(*
Searches an `I_Entity` for a `I_Receiver` component matching provided id pattern.
Result:
- Ok - Returns `I_Receiver`.
- None - Returns null.
- Err.Itf0 - Returns null, incorrect interface.
*)
FUNCTION GetReceiver : Result
VAR_INPUT
	iEntity		: I_Entity;
	sTagId		: Str;
END_VAR
VAR_OUTPUT
	iRec		: I_Receiver;
END_VAR
VAR
	i			: Iter(1);
	_iComp		: I_Component;
	cmp			: TagCmp;
END_VAR

IF iEntity = 0 THEN
	GetReceiver := Err.Itf0;
	RETURN;
END_IF

WHILE IsOk(iEntity.Get(i.Next(), iComp => _iComp)) DO
	IF IsOk(ICompToIRec(_iComp, iDest => iRec)) THEN
		IF cmp.Set(iRec.Tag).MatchWcdId(sTagId).IsTrue() THEN
			GetReceiver := Ok;
			RETURN;
		ELSE
			iRec := 0;
		END_IF
	END_IF
END_WHILE

END_FUNCTION

(* stored: Version 1.1.0.1
   POU GetReceiver: Id {7724b6ae-e8bc-4e18-87cf-f1d85e27fdd7}, SpecialFunc None *)
